Yaskawa INFORM job: R1_EMGPOUNCE.JBI

/JOB
//NAME R1_EMGPOUNCE
//POS
///NPOS 0,0,0,0,0,0
//INST
///DATE 2021/09/30 10:12
///ATTR SC,RW
///GROUP1 RB1
///LVARS 0,0,0,0,0,0,0,0
NOP
'%%%%%%%%%%%%%%%%%%%%%%%%%%%%%%%%
' R1 EMG Pounce Position
'%%%%%%%%%%%%%%%%%%%%%%%%%%%%%%%%
'
*TOP
'***********INITIALIZE***********
' Set Clear of Module Bits
CALL JOB:R1_CLEARMODULE ARGF234
' Report Position
CALL JOB:R1_REPORTPOS ARGF2
'********************************
'
'********PRE-STATUS_CHECK********
'********************************
'
'***********PRIME_MOVE***********
'********************************
MOVJ P[106] VJ=25.00
'
'*******POST-STATUS_CHECK********
'********************************
'
'****USER_DEFINED_PARAMETERS*****
'********************************
'
'********DATA_VALIDATION*********
'********************************
'
'*************SETUP**************
'********************************
'
'*************ACTION*************
'********************************
'
'*********HOUSE_KEEPING**********
CALL JOB:R1_CLEARMODULE ARGF999
SET B004 1
'********************************
*OUT
END
